// TIA Portal V16 export
// export: Created 2021-07-12T14:47:18.5799536Z, ExportSetting WithDefaults, DisplayName Totally Integrated Automation Portal, DisplayVersion V16, DisplayName TIA Portal Version Control Interface, DisplayVersion V16, DisplayName TIA Portal Openness, DisplayVersion V16, DisplayName STEP 7 Professional, DisplayVersion V16, DisplayName STEP 7 Safety, DisplayVersion V16, DisplayName WinCC Professional, DisplayVersion V16
TYPE "LSimaHydTO_typeForceControl"
TITLE = LSimaHydTO_typeForceControl
// Force control configuration data
// stored: IsFailsafeCompliant false
   STRUCT
      SmoothingTimeByChangeDifference { S7_SetPoint := 'True'} : LReal;   // Time constant for smoothing manipulated variable jumps
      PreControl { S7_SetPoint := 'True'} : LReal := 0.0;   // Weighting factor of the precontrol Kpc [%]
      Stiffness { S7_SetPoint := 'True'} : LReal;   // Stiffness of the system, should be > 0.0 if preControl is used
      ProportionalGain { S7_SetPoint := 'True'} : LReal := 1.0;   // Proportional gain Kp
      IntegralTime { S7_SetPoint := 'True'} : LReal;   // Active integral action time Ti [s]
      DerivativeTime { S7_SetPoint := 'True'} : LReal;   // Active derivative action time Td [s]
      DecayTime { S7_SetPoint := 'True'} : LReal := 0.0;   // Decay time constant of the DT1 component [s]
      OutputUppLimit { S7_SetPoint := 'True'} : LReal := 10000.0;   // Manipulated value high limit
      OutputLowLimit { S7_SetPoint := 'True'} : LReal := -10000.0;   // Manipulated value low limit
      SmoothSwitching { S7_SetPoint := 'True'} : Bool := TRUE;   // Switching mode to force control, if TRUE, initial command value of the force controller will be presetted for edgeless valve setpoint
      InvertSetpoint { S7_SetPoint := 'True'} : Bool;   // Invert output of controller if TRUE
   END_STRUCT;
END_TYPE
